Fanuc KAREL source: kt00439.KL

-- PROVISIONAL review KL for V1013-1; original PC SHA256 f9d3a648b8a992011813b2d8167ca0e9880918764343ac7086555ea3fccf74f3
-- Incomplete behavior may be omitted. Consult companion uncertainty JSON. Do not deploy.
PROGRAM KT00439
%NOLOCKGROUP
VAR
  I1 : INTEGER
  OUT : BOOLEAN
-- UNRESOLVED_DECL Y2 type=002018
BEGIN
  -- UNRESOLVED_PC offsets 5-16; opcodes 2E,23
  -- UNRESOLVED_PC offsets 21-35; opcodes 2E,22,9D,33,B2
  -- UNRESOLVED_PC offsets 40-62; opcodes 21,22,9D,33,B1,5C,23
  -- UNRESOLVED_PC offsets 67-71; opcodes 7F
END KT00439
